// Operated on linked list of type defined by T_DATA_TYPE Alias 
FUNCTION_BLOCK FB_Linked_List
VAR_INPUT
END_VAR
VAR_OUTPUT
END_VAR
VAR
	pHead :  POINTER TO ST_NODE;
	pTail :  POINTER TO ST_NODE;
END_VAR

// Creates/Adds an node to the end of the list
METHOD Create
VAR_INPUT
	Data : T_DATA_TYPE; // Data to add to new node.
END_VAR
VAR
	pTemp :  POINTER TO ST_NODE;
END_VAR
pTemp := __NEW(ST_NODE); 	// Allocate space in memory for a node.
pTemp^.Data := Data;		// Assign Data to the new node.
pTemp^.pNext := NULL;		// Pointer to next node is NULL.
IF pHead = 0 THEN pHead := pTemp; pTail := pTemp; // If the pointer to the pHead is NULL then give it an address. The pTail address of the first node is the pHead.
ELSE  pTail^.pNext := pTemp; pTail := pTail^.pNext; END_IF // Point previous node's pNext to the address of pTemp and set pTail to pTemp.
END_METHOD

// Empties/Clears/Deletes list
METHOD Empty
VAR
	pTemp : POINTER TO ST_NODE;
END_VAR
pTemp := pHead;
WHILE pTemp <> 0 DO
	pTemp := pTemp^.pNext; THIS^.Pop();
END_WHILE
END_METHOD

// Initializes or create an empty list
METHOD Init
pHead := NULL;
pTail := NULL;
END_METHOD

// Inserts node at a specific position in the list
METHOD Insert
VAR_INPUT
	Data 		: T_DATA_TYPE; 	// Data to add to new node.
	nPosition 	: UXINT;		// Position to add new node in list.
END_VAR
VAR
	pPrevious 	: POINTER TO ST_NODE;
	pCurrent 	: POINTER TO ST_NODE;
	pTemp 		: POINTER TO ST_NODE;
	i 			: UXINT;
END_VAR
pTemp := __NEW(ST_NODE);
pCurrent := pHead;
FOR i := 2 TO nPosition DO
	pPrevious := pCurrent;
	pCurrent := pPrevious^.pNext;
	END_FOR;
pTemp^.Data := Data;
pPrevious^.pNext := pTemp;
pTemp^.pNext := pCurrent;
END_METHOD

// Deletes/pops a node at the start of the list 
METHOD Pop
VAR
	pTemp : POINTER TO ST_NODE;
END_VAR
pTemp := pHead^.pNext;
__DELETE(pHead);
pHead := pTemp;
END_METHOD

// Adds/pushes a node at the start of the list 
METHOD Push
VAR_INPUT
	Data 	: T_DATA_TYPE;
END_VAR
VAR
	pTemp 	:  POINTER TO ST_NODE;
END_VAR
pTemp := __NEW(ST_NODE); 	// Allocate space in memory for a node.
pTemp^.Data := Data;
pTemp^.pNext := pHead;
pHead := pTemp;
END_METHOD

// Deletes node at a specific position in the list
METHOD Remove
VAR_INPUT
	nPosition 	: UXINT; // Position of node to delete.
END_VAR
VAR
	pPrevious 	: POINTER TO ST_NODE;
	pCurrent 	: POINTER TO ST_NODE;
	i 			: UXINT;
END_VAR
pCurrent := pHead;
FOR i := 2 TO nPosition DO
	pPrevious := pCurrent;
	pCurrent := pCurrent^.pNext;
	END_FOR;
pPrevious^.pNext := pCurrent^.pNext;
__DELETE(pCurrent);
END_METHOD

// Searches list for the first instance of data and returns it's location and whether it's in the list.
METHOD Search : BOOL
VAR_INPUT
	Data : T_DATA_TYPE; // Data to find in list
END_VAR
VAR_OUTPUT
	nPosition : UXINT; // Location of the data  starting from 1. 0 means data is not found in list
END_VAR
VAR
	pTemp 	: POINTER TO ST_NODE;
	i 		: UXINT;
END_VAR
pTemp := pHead;
FOR i := 1 TO THIS^.Size() DO
	Search := pTemp^.Data = Data;
	IF Search THEN nPosition := i; EXIT; ELSE nPosition := 0; END_IF
	pTemp := pTemp^.pNext;
	END_FOR
END_METHOD

// Traverse the list to display each node
METHOD Show
VAR_IN_OUT
	aList 		: ARRAY[*] OF T_DATA_TYPE; // Array to display data in list.
END_VAR
VAR
	pCurrent 	:  POINTER TO ST_NODE;
	i 			: DINT;
END_VAR
pCurrent := pHead;
i := LOWER_BOUND(aList, 1);
WHILE pCurrent <> 0 AND i < UPPER_BOUND(aList, 1) DO
	aList[i] := pCurrent^.Data;
	pCurrent := pCurrent^.pNext;
	i := i+1;
END_WHILE
END_METHOD

// Gets size of the list
METHOD Size : UXINT;
VAR
	pTemp 	: POINTER TO ST_NODE;
	i 		: UXINT;
END_VAR
pTemp := pHead;
WHILE pTemp <> 0 DO
	pTemp := pTemp^.pNext; i := i + 1;;
END_WHILE
Size := i;
END_METHOD

END_FUNCTION_BLOCK

(* stored: Version 1.1.0.1, ProductVersion 3.1.4024.4
   POU FB_Linked_List: Id {19223dee-072c-4cbb-9e58-eedc7741ea7e}, SpecialFunc None
   Method Create: Id {1c02436b-f1d7-46b9-bde8-e418c191c48f}
   Method Empty: Id {317ea86d-3d25-4a24-9aeb-8dd8eb13f3f4}
   Method Init: Id {d3845c5b-4488-4a2a-83ef-21fe8d01c1da}
   Method Insert: Id {b50ffa90-bffd-42d6-880d-1e20342d73fd}
   Method Pop: Id {a3623de3-4c8b-4ca0-a7a5-e2d659fad6d5}
   Method Push: Id {fc4a9c4f-82e1-46e6-8281-109c5a2f41f3}
   Method Remove: Id {e27d3464-0225-4467-9f8c-0a726d2728f5}
   Method Search: Id {da5f7172-2114-4eed-8448-2548351cb82a}
   Method Show: Id {44cc05c3-a73a-485e-b7c4-9f46d1a3c88e}
   Method Size: Id {cdf20009-0222-43c5-990c-054c16153aa7} *)
